// TIA Portal V19 export
FUNCTION_BLOCK "LiftCmd"   // FB11, LAD
TITLE = LiftCmd
{ S7_Optimized_Access := 'TRUE' }
AUTHOR : Siemens
// Lift command BeltLift
// stored: IsIECCheckEnabled true, MemoryReserve 100, SetENOAutomatically true
   VAR_INPUT
      interLockAuto { ExternalAccessible := 'False'; ExternalVisible := 'False'; ExternalWritable := 'False'} : Bool;   // Interlock automatic
      interLockMan { ExternalAccessible := 'False'; ExternalVisible := 'False'; ExternalWritable := 'False'} : Bool;   // Interlock manual
      autoStarted { ExternalAccessible := 'False'; ExternalVisible := 'False'; ExternalWritable := 'False'} : Bool;   // Automatic started
      autoLift { ExternalAccessible := 'False'; ExternalVisible := 'False'; ExternalWritable := 'False'} : "typeStartLift";   // Start auto lift
      manLift { ExternalAccessible := 'False'; ExternalVisible := 'False'; ExternalWritable := 'False'} : "typeStartLift";   // Start manual lift
      sensorLiftUp { ExternalAccessible := 'False'; ExternalVisible := 'False'; ExternalWritable := 'False'} : Bool;   // Sensor lift up
      sensorLiftDown { ExternalAccessible := 'False'; ExternalVisible := 'False'; ExternalWritable := 'False'} : Bool;   // Sensor lift down
   END_VAR
   VAR_OUTPUT
      liftUp { ExternalAccessible := 'False'; ExternalVisible := 'False'; ExternalWritable := 'False'} : Bool;   // Output lift up
      liftDown { ExternalAccessible := 'False'; ExternalVisible := 'False'; ExternalWritable := 'False'} : Bool;   // Output lift down
   END_VAR
   VAR
      statTrigLift { ExternalAccessible := 'False'; ExternalVisible := 'False'; ExternalWritable := 'False'} : "typeStartLift";   // Trigger lift up / Trigger lift
   END_VAR
BEGIN

REGION Network 1: set trigger lift up
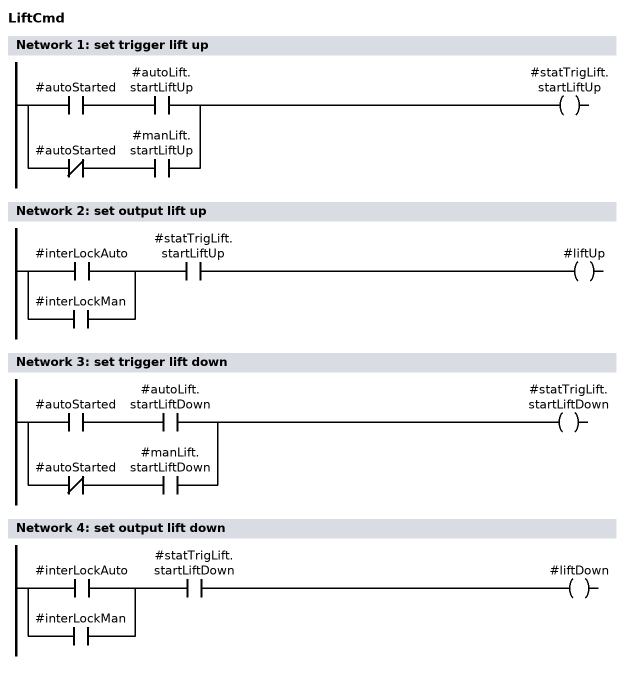
   RUNG wire#powerrail
      Contact( #autoStarted )
      Contact( #autoLift.startLiftUp )
      wire#w1
      Coil( #statTrigLift.startLiftUp )
   END_RUNG
   RUNG wire#powerrail
      I_Contact( #autoStarted )
      Contact( #manLift.startLiftUp )
   END_RUNG wire#w1
   // the same network as SCL:
   #statTrigLift.startLiftUp := (#autoStarted AND #autoLift.startLiftUp) OR (NOT #autoStarted AND #manLift.startLiftUp);
END_REGION

REGION Network 2: set output lift up
   RUNG wire#powerrail
      Contact( #interLockAuto )
      wire#w1
      Contact( #statTrigLift.startLiftUp )
      Coil( #liftUp )
   END_RUNG
   RUNG wire#powerrail
      Contact( #interLockMan )
   END_RUNG wire#w1
   // the same network as SCL:
   #liftUp := (#interLockAuto OR #interLockMan) AND #statTrigLift.startLiftUp;
END_REGION

REGION Network 3: set trigger lift down
   RUNG wire#powerrail
      Contact( #autoStarted )
      Contact( #autoLift.startLiftDown )
      wire#w1
      Coil( #statTrigLift.startLiftDown )
   END_RUNG
   RUNG wire#powerrail
      I_Contact( #autoStarted )
      Contact( #manLift.startLiftDown )
   END_RUNG wire#w1
   // the same network as SCL:
   #statTrigLift.startLiftDown := (#autoStarted AND #autoLift.startLiftDown) OR (NOT #autoStarted AND #manLift.startLiftDown);
END_REGION

REGION Network 4: set output lift down
   RUNG wire#powerrail
      Contact( #interLockAuto )
      wire#w1
      Contact( #statTrigLift.startLiftDown )
      Coil( #liftDown )
   END_RUNG
   RUNG wire#powerrail
      Contact( #interLockMan )
   END_RUNG wire#w1
   // the same network as SCL:
   #liftDown := (#interLockAuto OR #interLockMan) AND #statTrigLift.startLiftDown;
END_REGION
END_FUNCTION_BLOCK
